// TIA Portal V19 export
DATA_BLOCK "faceplate_DB_2"   // DB4
// stored: InstanceOfName faceplate, InstanceOfType FB
"faceplate"
   // VAR_INPUT
   //    start : Bool;
   //    stop : Bool;
   // END_VAR
   // VAR_OUTPUT
   //    "conveyor-right" : Bool;
   //    "conveyor-left" : Bool;
   // END_VAR
   // VAR_IN_OUT
   //    "Time-Right" : Time;
   //    "Time-Right-Rest" : Time;
   //    "Time-Left" : Time;
   //    "Time-Left-Rest" : Time;
   //    "memory-stop" : Bool;
   //    "memory-start" : Bool;
   //    "Timer-Right" : TP_TIME;
   //    "Timer-Right-Rest" : TP_TIME;
   //    "Timer-Left" : TP_TIME;
   //    "Timer-Left-Rest" : TP_TIME;
   // END_VAR
   // VAR
   //    "mem-start" : Bool;
   //    "mem-stop" : Bool;
   //    "mem-edge-1" : Bool;
   //    "mem-edge-2" : Bool;
   //    "mem-edge-3" : Bool;
   //    "mem-edge-4" : Bool;
   //    "mem-edge-5" : Bool;
   //    "mem-edge-6" : Bool;
   // END_VAR
BEGIN
END_DATA_BLOCK
